FUNCTION ReplaceString
VAR_INPUT
	in : ANY;
	replaced : T_MaxString;
	with : T_MaxString;
END_VAR
VAR
	replaceBegin : UDINT;
END_VAR

replaceBegin := FIND2(in.pValue, ADR(replaced));

IF (replaceBegin = 0) THEN
	RETURN;
END_IF

REPLACE2(in.pValue, ADR(with), in.pValue, TO_UDINT(in.diSize), TO_UDINT(LEN(replaced)), replaceBegin);

END_FUNCTION

(* stored: Version 1.1.0.1
   POU ReplaceString: Id {1d9a911a-d2c2-41a5-bc59-e93c9a23e24a}, SpecialFunc None *)
